(*			
	EVERDE sp. z o.o.
	Rafał Osajda		22.01.2025		TC 4026.13		wer. 0.0.0.1
	B_Baza dla czujników binarnych 	
*)
FUNCTION_BLOCK ABSTRACT FB_IOSensor EXTENDS FB_BaseComponent IMPLEMENTS ITF_IOSensor, ITF_IOSensor_HMI_Init
VAR
	bContact				AT %I*	: BOOL;		// Styk czujnika
	eType							: E_IOSensorType;
END_VAR

METHOD PUBLIC GetSensorType : E_IOSensorType
VAR_INPUT
END_VAR
GetSensorType			:= THIS^.eType;
END_METHOD

METHOD PUBLIC GetSensorTypeToString : STRING
VAR CONSTANT
	arrType		: ARRAY [0..2] OF STRING := ['NO', 'NC', 'NOx2'];
END_VAR
GetSensorTypeToString			:= arrType [TO_INT (THIS^.eType)];
END_METHOD

(*			
	EVERDE sp. z o.o.
	Rafał Osajda		05.02.2025		TC 4026.13		wer. 0.0.0.1
	Zwraca aktualny stan czujnika
*)
METHOD IsActive : BOOL
END_METHOD

END_FUNCTION_BLOCK

(* stored: Version 1.1.0.1
   POU FB_IOSensor: Id {38d74651-ddd4-440f-81aa-c82978b08fa3}, SpecialFunc None
   Method GetSensorType: Id {f374bc07-fad7-40f2-bc55-235455285601}
   Method GetSensorTypeToString: Id {4ad723da-d327-4de9-9137-959624f49814}
   Method IsActive: Id {db6dccc1-2a7a-463e-864e-da1a3729b042} *)
